Yaskawa INFORM job: SVETS.JBI

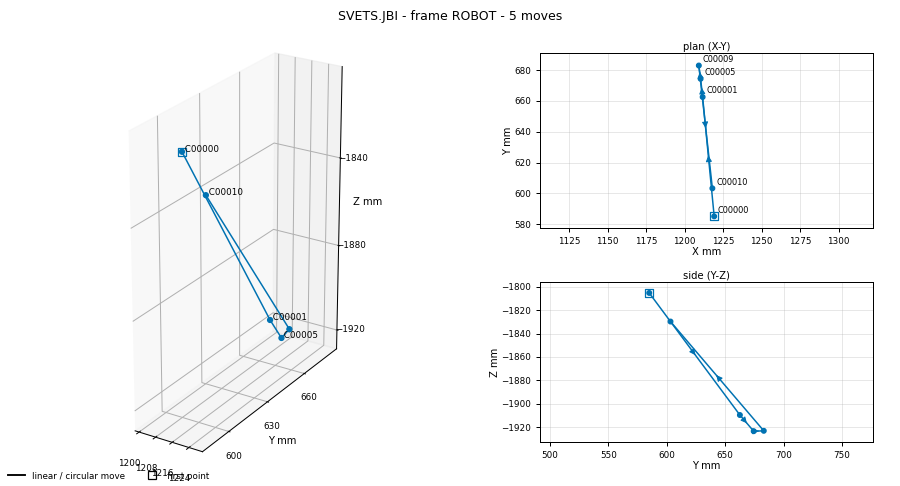
[picture p0: tool path of SVETS.JBI in frame ROBOT, 5 of 5 moves have a stored position in this frame; points joined in program order, loops and branches not executed]
/JOB
//NAME SVETS
///FOLDERNAME INNE
//POS
///NPOS 11,11,0,1,0,0
///TOOL 0
///POSTYPE ROBOT
///RECTAN
///RCONF 0,0,0,0,1,0,0,0,0,0,0,0,0,0,0,0,0,0,0,0,0,0,0,0
C00000=1219.225,585.030,-1805.251,40.6411,-1.1292,7.6176
C00001=1211.726,662.575,-1909.670,40.6455,-1.1278,7.6123
C00002=1211.726,662.575,-1909.670,40.6455,-1.1278,7.6123
C00003=1211.765,674.656,-1909.674,40.6444,-1.1296,7.6111
C00004=1211.728,662.569,-1923.475,40.6445,-1.1282,7.6129
C00005=1210.410,674.391,-1923.512,40.6454,-1.1279,7.6131
C00006=1210.400,674.386,-1896.163,40.6450,-1.1275,7.6131
C00007=1210.412,637.973,-1923.522,40.6435,-1.1301,7.6151
C00008=1209.243,683.022,-1923.176,40.6452,-1.1275,7.6151
C00009=1209.243,683.022,-1923.176,40.6452,-1.1275,7.6151
C00010=1218.053,603.234,-1829.714,40.6445,-1.1272,7.6159
///RCONF 0,0,0,0,0,0,0,0,0,0,0,0,0,0,0,0,0,0,0,0,0,0,0,0
BC00000=1.890,2751.820,818.150
BC00001=1.890,2751.820,818.150
BC00002=1.890,2751.820,818.150
BC00003=1.890,2751.820,818.150
BC00004=1.890,2751.820,818.150
BC00005=1.890,2751.820,818.150
BC00006=1.890,2751.820,818.150
BC00007=1.890,2751.820,818.150
BC00008=269.302,2751.820,818.150
BC00009=269.302,2751.820,818.150
BC00010=269.302,2751.820,818.150
///RCONF 0,0,0,0,1,0,0,0,0,0,0,0,0,0,0,0,0,0,0,0,0,0,0,0
P00010=-0.015,0.468,-0.695,0.0000,0.0000,0.0000
//INST
///DATE 2023/10/04 15:16
///ATTR SC,RW,RJ
////FRAME ROBOT
///GROUP1 RB1,BS1
NOP
SFTOF
MOVL C00000 BC00000 V=150.0
MACRO1 MJ#(0) ARGF3
MOVL C00001 BC00001 V=75.0
REFP 4 C00002 BC00002
REFP 5 C00003 BC00003
REFP 6 C00004 BC00004
CALL JOB:SRCH-2D-R1
SFTON P010
MOVL C00005 BC00005 V=75.0
REFP 1 C00006 BC00006
REFP 2 C00007 BC00007
REFP 3 C00008 BC00008
ARCON
WVON WEV#(1)
MOVL C00009 BC00009 V=7.5
WVOF
ARCOF
SFTOF
MOVL C00010 BC00010 V=150.0
END
